(* PLC project rangesensor, Dassault Systèmes ControlBuild 2024x *)
(* stored: creationDateTime 2023-10-03T11:13:55-01:00 *)

(* This module simulates the behaviour of an over threshold sensor with a detection area. *)
FUNCTION_BLOCK tri_chain.rangesensor
  VAR_INPUT
    level : REAL := 0.0;
    sensorSupply : BOOL := true;
  END_VAR
  VAR_OUTPUT
    rangeSensor : BOOL := false;
  END_VAR
  VAR
    status_act_prod : DINT := 0;
    m11 : REAL := 1.0;
    m12 : REAL := 0.0;
    m13 : REAL := 0.0;
    m14 : REAL := 0.0;
    m21 : REAL := 0.0;
    m22 : REAL := 1.0;
    m23 : REAL := 0.0;
    m24 : REAL := 0.0;
    m31 : REAL := 0.0;
    m32 : REAL := 0.0;
    m33 : REAL := 1.0;
    m34 : REAL := 0.0;
    m41 : REAL := 0.0;
    m42 : REAL := 0.0;
    m43 : REAL := 0.0;
    m44 : REAL := 1.0;
  END_VAR
  VAR CONSTANT
    threshold : REAL := 500.0;
    range : REAL := 10.0;
    wiringLogic : BOOL := true;
  END_VAR
  VAR
    d_sensor : BOOL := false;
    v_d_sensor : BOOL := false;
  END_VAR


ACTION C_source_code:
/* ----------------------------------------------------------------	*/
/* Type : Model of Operative Behaviour					*/
/* Category :  Sensors							*/
/* Author : Dassault Systemes						*/
/* Update date : June 2018							*/
/* ----------------------------------------------------------------	*/
/* This module simulates the behaviour 					*/
/* of an over threshold sensor with a detection area.			*/
/* ----------------------------------------------------------------	*/
/* In the case of a faulty element, it takes the fault value else 	*/
/* it takes the state of the sensor in function of its wiring logic.	*/ 
/* ----------------------------------------------------------------	*/

if (d_sensor) rangeSensor = v_d_sensor;
else
	if ( sensorSupply ) rangeSensor = ((level >= threshold) & (level <= (threshold + range))) ^ ! wiringLogic;
	else rangeSensor = 0;
END_ACTION
END_FUNCTION_BLOCK
